{attribute 'GeneratedUsingTerminal: EPP1518-0002-0016'}
{attribute addProperty BoxType "EPP1518-0002-0016"}
{attribute addProperty Id "StatusAT %I*Status_57491DF17Counter_valueAT %I*UDINT4"}
{attribute addProperty CRC "4279287100"}
{attribute addProperty Size "11"}
TYPE CNT_Input_Channel_FF10BD3C EXTENDS InputBase_8311D824 :
STRUCT
	{attribute addProperty Name "Status"}
	Status AT %I* : Status_57491DF1;
	{attribute addProperty Name "Counter_value"}
	Counter_value AT %I* : UDINT;
END_STRUCT
END_TYPE

(* stored: Version 1.2.0.0, ProductVersion 3.1.4024.11
   DUT CNT_Input_Channel_FF10BD3C: Id {f5714c3d-fc18-4c1a-b36b-52b8154db615} *)
